FUNCTION_BLOCK Label IMPLEMENTS I_Label
VAR
	_label AT%M* : T_MaxString;
END_VAR

PROPERTY Text : STRING
GET
Text := _label;
END_GET
SET
_label := Text;
END_SET
END_PROPERTY

END_FUNCTION_BLOCK

(* stored: Version 1.1.0.1, ProductVersion 3.1.4024.12
   POU Label: Id {01cd52d5-6d31-4fef-badc-d3b37de77d96}, SpecialFunc None
   Property Text: Id {5d28d2d3-eec5-4f47-a2c0-c633c36293d2}
   Get Get: Id {2724fdfa-d80d-43c0-b130-c6ac5b808dd9}
   Set Set: Id {b30128c3-69fe-43af-8ada-98f61467938f} *)
